Yaskawa INFORM job: INIT_ROS.JBI

/JOB
//NAME INIT_ROS
//POS
///NPOS 0,0,0,0,0,0
//INST
///DATE 2014/06/16 21:00
///ATTR SC,RW
///GROUP1 RB2,BS2
///GROUP2 RB1,BS1
NOP
DOUT OT#(890) OFF
DOUT OT#(889) OFF
TIMER T=0.050
DOUT OT#(889) ON
WAIT OT#(890)=ON
DOUT OT#(890) OFF
END
